Staubli VAL3: initSensor.pgx

public program initSensor(string& x_sSocket, FlagStatus& x_fSensorStatus)
  local num l_nSensorReturn[4]
  local num l_nNum
  local num l_nReturn
  local num l_nFilter
  local num l_nSensitivity[49]
  local string l_sValue[49]
  local string l_sString
  local bool l_bReport
  local num l_nSampleSum[6]
  local num l_nSampleData[6]
  local num SampleNum
begin

  //This program is used for initializing the Force/Torque sensor settings and connecting the sensor to the
  //robot controller.


  //Define the socket communication parameter for the Force/Torque sensor
  cSensorCommParm.port=5001
  cSensorCommParm.timeOut=5
  cSensorCommParm.mode="rs422"
  cSensorCommParm.nagle=false
  //Configure the socket communication parameter for the Force/Torque sensor
  l_nReturn=getData(x_sSocket,sClientSensor)
  if l_nReturn>0
    l_nSensorReturn[0]=sioCtrl(sClientSensor,"port",cSensorCommParm.port)
    l_nSensorReturn[1]=sioCtrl(sClientSensor,"timeout",cSensorCommParm.timeOut)
    l_nSensorReturn[2]=sioCtrl(sClientSensor,"mode",cSensorCommParm.mode)
    l_nSensorReturn[3]=sioCtrl(sClientSensor,"nagle",cSensorCommParm.nagle)
  endIf
  //Check the socket communication configuration successful or not
  //if (l_nSensorReturn[0]==0) and (l_nSensorReturn[1]==0) and (l_nSensorReturn[2]==0) and (l_nSensorReturn[3]==0)
  if l_nSensorReturn==0
    x_fSensorStatus.ForceFlag=1
  else
    x_fSensorStatus.ForceFlag=-1
  endIf

  //Acquire and Configure the Force/Torque sensor(Wacoh) relevant functional parameters
  //Acquire the moving average filter settings of Wacoh sensor
  sClientSensor="0F"
  clearBuffer(sClientSensor)
  sioGet(sClientSensor,l_nFilter)
  //Configrue the moving average filter settings to 250Hz for synchronizing the robot motion in every 4ms
  if l_nFilter==52
    putln("Filter setting is ok!")
    delay(0.5)
  else
    sClientSensor="4F"
    putln("Filter setting is wrong, but changed correctly!")
    delay(0.5)
  endIf

  //Acquire and store the sensitivity of the Wacoh sensor
  //Acquire the sensitivity of the sensor in lowercase p command
  sClientSensor="p"
  clearBuffer(sClientSensor)
  sioGet(sClientSensor,l_nSensitivity)
  //Convert the decimal text to the number and store it in the public array nSensitivity
  for l_nNum=0 to 46
    l_sValue[l_nNum]=chr(l_nSensitivity[l_nNum])
    l_sString=l_sString+l_sValue[l_nNum]
  endFor
  //Display the Wacoh sensor sensitivity
  putln(l_sString)
  for l_nNum=0 to 5
    l_sString=toNum(l_sString,nSensitivity[l_nNum],l_bReport)
  endFor

  //Reset the offset of the Wacoh sensor for several times every time the sensor will be used
  l_nNum=0
  do
    sClientSensor="O"
    l_nNum=l_nNum+1
  until l_nNum==10

  //Acquire the zero point of the Wacoh sensor with endeffector based on sampling for lower random noise error
  l_nSampleSum=0
  SampleNum=0
  do
    call readDetectValue(l_nSampleData,x_fSensorStatus)
    for l_nNum=0 to 5
      l_nSampleSum[l_nNum]=l_nSampleSum[l_nNum]+l_nSampleData[l_nNum]
    endFor
    SampleNum=SampleNum+1
  until SampleNum==200
  //Store the zero point of the Wacoh sensor in the public array
  for l_nNum=0 to 5
    nZeroPoint[l_nNum]=l_nSampleSum[l_nNum]/SampleNum
  endFor

  delay(0.0)

end
